INTERFACE I_Actuator EXTENDS I_Device

METHOD Start : bool
VAR_INPUT
END_VAR
END_METHOD

METHOD Stop : bool
VAR_INPUT
END_VAR
END_METHOD

END_INTERFACE

(* stored: Version 1.1.0.1
   Itf I_Actuator: Id {ee4b77db-2f06-45ab-acc6-e79bd2b64c95}
   Method Start: Id {0696696c-f68d-49af-b839-36eaf39c0aa7}
   Method Stop: Id {b02047bc-d8d7-4e58-8220-ea5b2536317c} *)
